FUNCTION_BLOCK TEvent_MinutesChanged EXTENDS TEventBase IMPLEMENTS IEvent
VAR
	Now: TIMESTRUCT;
    Handler : IEventHandler_OnMinutesChanged;
END_VAR

METHOD  CallHandler
VAR_INPUT
    HandlerBase : IEventHandlerBase;
END_VAR
IF __QUERYINTERFACE(HandlerBase,Handler) THEN
    Handler.OnMinutesChanged(Now);
END_IF
END_METHOD

METHOD  IsHandlerSupported : BOOL
VAR_INPUT
    EventHandler : IEventHandlerBase;
END_VAR
IF __QUERYINTERFACE(EventHandler,Handler) THEN
    IsHandlerSupported := TRUE;
END_IF
END_METHOD

METHOD RaiseEx
VAR_INPUT
	Now: TIMESTRUCT;
END_VAR
THIS^.Now := Now;
SUPER^.Raise();
END_METHOD

END_FUNCTION_BLOCK

(* stored: Version 1.1.0.1, ProductVersion 3.1.4024.3
   POU TEvent_MinutesChanged: Id {012c5b9e-1d8a-0f45-0078-62e7532178fc}, SpecialFunc None
   Method CallHandler: Id {278a7906-30ee-09c5-0407-481845d076bf}
   Method IsHandlerSupported: Id {d56163f5-7fc3-0d4f-29b3-87e7475083df}
   Method RaiseEx: Id {0db731e5-9bc7-0aeb-30bf-2e83a1cb0981} *)
